// TIA Portal project "Palletizer" (V15.1)

(* hardware
DEVICE "S71500/ET200MP-Station_1"  S7-1500 station
   slot 0: "Profilschiene_0"  6ES7 590-1***0-0AA0
   slot 1: "PLC_1"  CPU 1511-1 PN  6ES7 511-1AK00-0AB0  V1.8
   slot 2: "AI 8xU/I/RTD/TC ST_1"  AI 8xU/I/RTD/TC ST  6ES7 531-7KF00-0AB0  V2.0
   slot 3: "AI 8xU/I/RTD/TC ST_2"  AI 8xU/I/RTD/TC ST  6ES7 531-7KF00-0AB0  V2.0
   slot 4: "AI 8xU/I/RTD/TC ST_3"  AI 8xU/I/RTD/TC ST  6ES7 531-7KF00-0AB0  V2.0
   slot 5: "AI 8xU/I/RTD/TC ST_4"  AI 8xU/I/RTD/TC ST  6ES7 531-7KF00-0AB0  V2.0
   slot 6: "DI 16x24VDC BA_1"  DI 16x24VDC BA  6ES7 521-1BH10-0AA0  V1.0
*)

// ===== PLC "PLC_1"  CPU 1511-1 PN =====

VAR_GLOBAL   // PLC tag table "Standard-Variablentabelle"
   "Pallet at entry" AT %E0.0 : Bool;
   "Clock_Byte" AT %MB0 : Byte;
   "Clock_10Hz" AT %M0.0 : Bool;
   "Clock_5Hz" AT %M0.1 : Bool;
   "Clock_2.5Hz" AT %M0.2 : Bool;
   "Clock_2Hz" AT %M0.3 : Bool;
   "Clock_1.25Hz" AT %M0.4 : Bool;
   "Clock_1Hz" AT %M0.5 : Bool;
   "Clock_0.625Hz" AT %M0.6 : Bool;
   "Clock_0.5Hz" AT %M0.7 : Bool;
   "Pallet at exit" AT %I0.1 : Bool;
   "Pallet loaded" AT %I0.2 : Bool;
   "Box at entry" AT %I0.3 : Bool;
   "Pusher at limit" AT %I0.4 : Bool;
   "Plate limit" AT %I0.5 : Bool;
   "Clamped" AT %I0.6 : Bool;
   "Elevator moving" AT %I0.7 : Bool;
   "Start" AT %I1.0 : Bool;
   "Reset" AT %I1.1 : Bool;
   "Stop" AT %I1.2 : Bool;
   "Emergency stop" AT %I1.3 : Bool;
   "Auto" AT %I1.4 : Bool;
   "Pallet feeder" AT %Q0.0 : Bool;
   "Laod pallet" AT %Q0.1 : Bool;
   "Exit conveyor" AT %Q0.2 : Bool;
   "Move to limit" AT %Q0.3 : Bool;
   "Elevator up" AT %Q0.4 : Bool;
   "Elevator down" AT %Q0.5 : Bool;
   "Box feeder" AT %Q0.6 : Bool;
   "Turn" AT %Q0.7 : Bool;
   "Push" AT %Q1.0 : Bool;
   "Load belt" AT %Q1.1 : Bool;
   "Clamp" AT %Q1.2 : Bool;
   "Open plate" AT %Q1.3 : Bool;
   "Warning light" AT %Q1.4 : Bool;
   "Start light" AT %Q1.5 : Bool;
   "Reset light" AT %Q1.6 : Bool;
   "Stop light" AT %Q1.7 : Bool;
   "Counter" AT %QD30 : DInt;
END_VAR

TYPE "statusCiclo"
   STRUCT
      EmAutomatico : Bool;
      EmManual : Bool;
      CicloIniciado : Bool;
      EmAnomalia : Bool;
      EmEmergencia : Bool;
      EmParada : Bool;
      Reset : Bool;
      AddCont : DInt;
   END_STRUCT;
END_TYPE

TYPE "Controle_Caixas"
   STRUCT
      N_Caixas : Int;
      N_Atingido : Bool;
      Solicitacao_Box : Bool;
      Reset_N_Caixas : Bool;
      Aux_Ordenacao : Bool;
      Ordenado : Bool;
   END_STRUCT;
END_TYPE

// folder: Paletizador

DATA_BLOCK "Painel_DB"   // DB1
{ S7_Optimized_Access := 'TRUE' }
VERSION : 0.1
// stored: InstanceOfName Painel
"Painel"
BEGIN
END_DATA_BLOCK

DATA_BLOCK "Pallet_Feeder_DB"   // DB2
{ S7_Optimized_Access := 'TRUE' }
VERSION : 0.1
// stored: InstanceOfName Pallet_Feeder
"Pallet_Feeder"
BEGIN
END_DATA_BLOCK

DATA_BLOCK "Status"   // DB3
{ S7_Optimized_Access := 'TRUE' }
VERSION : 0.1
BEGIN
END_DATA_BLOCK

DATA_BLOCK "Remove_Pallet_DB"   // DB4
{ S7_Optimized_Access := 'TRUE' }
VERSION : 0.1
// stored: InstanceOfName Remove_Pallet
"Remove_Pallet"
BEGIN
END_DATA_BLOCK

DATA_BLOCK "Box_Feeder_DB"   // DB5
{ S7_Optimized_Access := 'TRUE' }
VERSION : 0.1
// stored: InstanceOfName Box_Feeder
"Box_Feeder"
BEGIN
END_DATA_BLOCK

DATA_BLOCK "Elevador_DB"   // DB6
{ S7_Optimized_Access := 'TRUE' }
VERSION : 0.1
// stored: InstanceOfName Elevador
"Elevador"
BEGIN
END_DATA_BLOCK

DATA_BLOCK "Organizador_DB"   // DB7
{ S7_Optimized_Access := 'TRUE' }
VERSION : 0.1
// stored: InstanceOfName Organizador
"Organizador"
BEGIN
END_DATA_BLOCK

// folder: Paletizador/Organizador

DATA_BLOCK "Orientacao_2_DB"   // DB8
{ S7_Optimized_Access := 'TRUE' }
VERSION : 0.1
// stored: InstanceOfName Orientacao_2
"Orientacao_2"
BEGIN
END_DATA_BLOCK

DATA_BLOCK "Orientacao_1_DB"   // DB10
{ S7_Optimized_Access := 'TRUE' }
VERSION : 0.1
// stored: InstanceOfName Orientacao_1
"Orientacao_1"
BEGIN
END_DATA_BLOCK

// folder: System blocks/Program resources

DATA_BLOCK "Contadir_Camadas"   // DB9
{ S7_Optimized_Access := 'TRUE' }
AUTHOR : Simatic
FAMILY : IEC
NAME : CNTR
VERSION : 1.0
// stored: InstanceOfName IEC_COUNTER
"IEC_COUNTER"
BEGIN
END_DATA_BLOCK

DATA_BLOCK "Contador_Caixas"   // DB11
{ S7_Optimized_Access := 'TRUE' }
AUTHOR : Simatic
FAMILY : IEC
NAME : CNTR
VERSION : 1.0
// stored: InstanceOfName IEC_COUNTER
"IEC_COUNTER"
BEGIN
END_DATA_BLOCK

DATA_BLOCK "Timer_Load_Belt"   // DB13
{ S7_Optimized_Access := 'TRUE' }
AUTHOR : Simatic
FAMILY : IEC
NAME : IEC_TMR
VERSION : 1.0
// stored: InstanceOfName IEC_TIMER
"IEC_TIMER"
BEGIN
END_DATA_BLOCK

DATA_BLOCK "Counter_Push"   // DB14
{ S7_Optimized_Access := 'TRUE' }
AUTHOR : Simatic
FAMILY : IEC
NAME : CNTR
VERSION : 1.0
// stored: InstanceOfName IEC_COUNTER
"IEC_COUNTER"
BEGIN
END_DATA_BLOCK

DATA_BLOCK "Ton_Reset_Push"   // DB15
{ S7_Optimized_Access := 'TRUE' }
AUTHOR : Simatic
FAMILY : IEC
NAME : IEC_TMR
VERSION : 1.0
// stored: InstanceOfName IEC_TIMER
"IEC_TIMER"
BEGIN
END_DATA_BLOCK

DATA_BLOCK "Timer_Clamp"   // DB16
{ S7_Optimized_Access := 'TRUE' }
AUTHOR : Simatic
FAMILY : IEC
NAME : IEC_TMR
VERSION : 1.0
// stored: InstanceOfName IEC_TIMER
"IEC_TIMER"
BEGIN
END_DATA_BLOCK

DATA_BLOCK "Timer_Desce"   // DB17
{ S7_Optimized_Access := 'TRUE' }
AUTHOR : Simatic
FAMILY : IEC
NAME : IEC_TMR
VERSION : 1.0
// stored: InstanceOfName IEC_TIMER
"IEC_TIMER"
BEGIN
END_DATA_BLOCK

// folder: (top level)

FUNCTION "MHJ-PLC-Lab-Function-S71500" : Void   // FC9000, SCL
{ S7_Optimized_Access := 'TRUE' }
VERSION : 0.1
   VAR_TEMP
      Value : Byte;
      ForCounter : Int;
   END_VAR
   VAR CONSTANT
      Value_01_DW : DWord := 16#1223_5486;
      Value_02_DW : DWord := 16#A6C9_D1F5;
   END_VAR
BEGIN

   #Value:=PEEK(area := 16#82,
        dbNumber := 0,
        byteOffset := 511);
   #Value := #Value + 1;

   POKE(area := 16#82,
        dbNumber := 0,
        byteOffset := 511,
        value := #Value);

   POKE(area := 16#82,
        dbNumber := 0,
        byteOffset := 1016,
        value := #Value_01_DW);
   POKE(area := 16#82,
        dbNumber := 0,
        byteOffset := 1020,
        value := #Value_02_DW);

   FOR #ForCounter := 0 TO 63 DO
       #Value:=PEEK(area := 16#1,
            dbNumber := 0,
            byteOffset := #ForCounter);
       POKE(area := 16#81,
            dbNumber := 0,
            byteOffset := #ForCounter,
            value := #Value);
   END_FOR;
   #Value := PEEK(area := 16#1,
                  dbNumber := 0,
                  byteOffset := 512);
   POKE(area := 16#82,
        dbNumber := 0,
        byteOffset := 512,
        value := #Value);
END_FUNCTION

ORGANIZATION_BLOCK "Main"   // OB1, FBD, ProgramCycle
TITLE = "Main Program Sweep (Cycle)"
{ S7_Optimized_Access := 'TRUE' }
VERSION : 0.1
   VAR_INPUT
      Initial_Call : Bool;   // Initial call of this OB
      Remanence : Bool;   // =True, if remanent data are available
   END_VAR
BEGIN

REGION Network 1
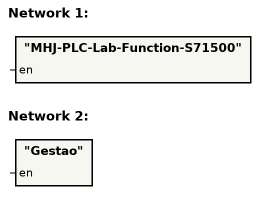
   "MHJ-PLC-Lab-Function-S71500"();
END_REGION

REGION Network 2
   "Gestao"();
END_REGION
END_ORGANIZATION_BLOCK

// folder: Paletizador

FUNCTION "Gestao" : Void   // FC1, LAD
{ S7_Optimized_Access := 'TRUE' }
VERSION : 0.1
BEGIN

REGION Network 1
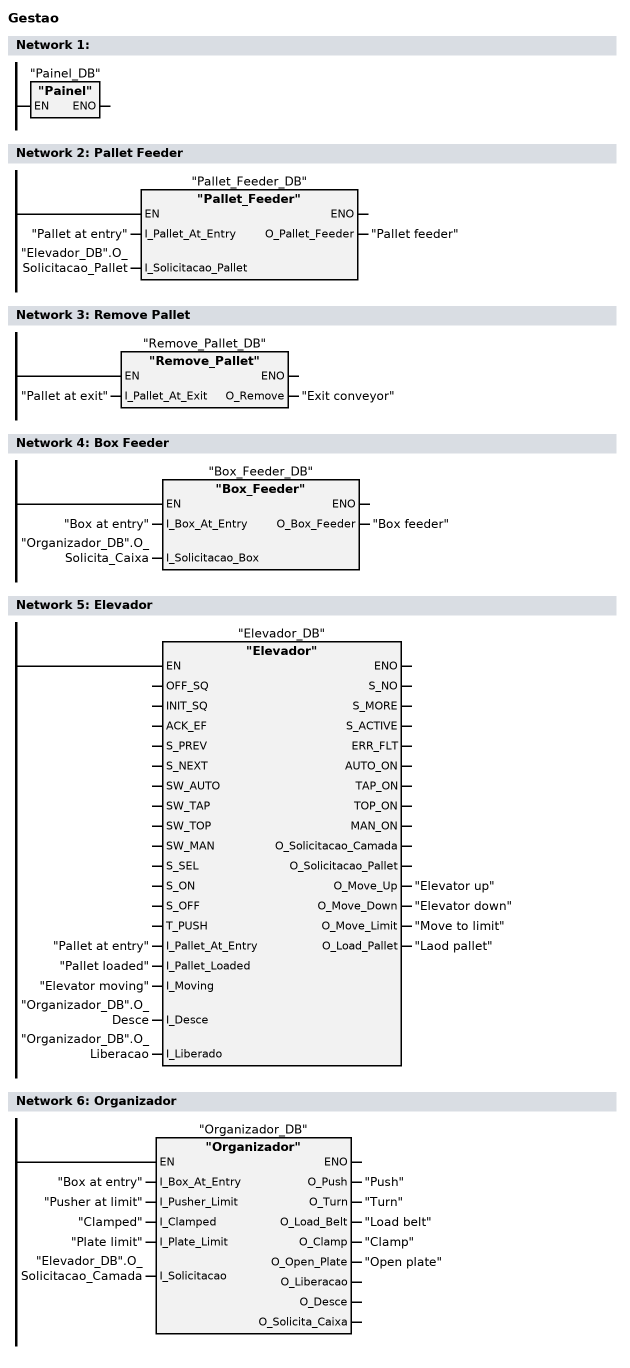
   RUNG wire#powerrail
      "Painel_DB"()
   END_RUNG
   // the same network as SCL:
   "Painel_DB"();   // "Painel"
END_REGION

REGION Network 2: Pallet Feeder
   RUNG wire#powerrail
      "Pallet_Feeder_DB"(I_Pallet_At_Entry := "Pallet at entry", I_Solicitacao_Pallet := "Elevador_DB".O_Solicitacao_Pallet, O_Pallet_Feeder => "Pallet feeder")
   END_RUNG
   // the same network as SCL:
   "Pallet_Feeder_DB"(I_Pallet_At_Entry := "Pallet at entry",   // "Pallet_Feeder"
                      I_Solicitacao_Pallet := "Elevador_DB".O_Solicitacao_Pallet,
                      O_Pallet_Feeder => "Pallet feeder");
END_REGION

REGION Network 3: Remove Pallet
   RUNG wire#powerrail
      "Remove_Pallet_DB"(I_Pallet_At_Exit := "Pallet at exit", O_Remove => "Exit conveyor")
   END_RUNG
   // the same network as SCL:
   "Remove_Pallet_DB"(I_Pallet_At_Exit := "Pallet at exit", O_Remove => "Exit conveyor");   // "Remove_Pallet"
END_REGION

REGION Network 4: Box Feeder
   RUNG wire#powerrail
      "Box_Feeder_DB"(I_Box_At_Entry := "Box at entry", I_Solicitacao_Box := "Organizador_DB".O_Solicita_Caixa, O_Box_Feeder => "Box feeder")
   END_RUNG
   // the same network as SCL:
   "Box_Feeder_DB"(I_Box_At_Entry := "Box at entry",   // "Box_Feeder"
                   I_Solicitacao_Box := "Organizador_DB".O_Solicita_Caixa,
                   O_Box_Feeder => "Box feeder");
END_REGION

REGION Network 5: Elevador
   RUNG wire#powerrail
      "Elevador_DB"(OFF_SQ :=, INIT_SQ :=, ACK_EF :=, S_PREV :=, S_NEXT :=, SW_AUTO :=, SW_TAP :=, SW_TOP :=, SW_MAN :=, S_SEL :=, S_ON :=, S_OFF :=, T_PUSH :=, I_Pallet_At_Entry := "Pallet at entry", I_Pallet_Loaded := "Pallet loaded", I_Moving := "Elevator moving", I_Desce := "Organizador_DB".O_Desce, I_Liberado := "Organizador_DB".O_Liberacao, S_NO =>, S_MORE =>, S_ACTIVE =>, ERR_FLT =>, AUTO_ON =>, TAP_ON =>, TOP_ON =>, MAN_ON =>, O_Solicitacao_Camada =>, O_Solicitacao_Pallet =>, O_Move_Up => "Elevator up", O_Move_Down => "Elevator down", O_Move_Limit => "Move to limit", O_Load_Pallet => "Laod pallet")
   END_RUNG
   // the same network as SCL:
   "Elevador_DB"(I_Pallet_At_Entry := "Pallet at entry",   // "Elevador"
                 I_Pallet_Loaded := "Pallet loaded",
                 I_Moving := "Elevator moving",
                 I_Desce := "Organizador_DB".O_Desce,
                 I_Liberado := "Organizador_DB".O_Liberacao,
                 O_Move_Up => "Elevator up",
                 O_Move_Down => "Elevator down",
                 O_Move_Limit => "Move to limit",
                 O_Load_Pallet => "Laod pallet");
END_REGION

REGION Network 6: Organizador
   RUNG wire#powerrail
      "Organizador_DB"(I_Box_At_Entry := "Box at entry", I_Pusher_Limit := "Pusher at limit", I_Clamped := "Clamped", I_Plate_Limit := "Plate limit", I_Solicitacao := "Elevador_DB".O_Solicitacao_Camada, O_Push => "Push", O_Turn => "Turn", O_Load_Belt => "Load belt", O_Clamp => "Clamp", O_Open_Plate => "Open plate", O_Liberacao =>, O_Desce =>, O_Solicita_Caixa =>)
   END_RUNG
   // the same network as SCL:
   "Organizador_DB"(I_Box_At_Entry := "Box at entry",   // "Organizador"
                    I_Pusher_Limit := "Pusher at limit",
                    I_Clamped := "Clamped",
                    I_Plate_Limit := "Plate limit",
                    I_Solicitacao := "Elevador_DB".O_Solicitacao_Camada,
                    O_Push => "Push",
                    O_Turn => "Turn",
                    O_Load_Belt => "Load belt",
                    O_Clamp => "Clamp",
                    O_Open_Plate => "Open plate");
END_REGION
END_FUNCTION

// folder: Paletizador/Box_Feeder

FUNCTION_BLOCK "Box_Feeder"   // FB4, LAD
{ S7_Optimized_Access := 'TRUE' }
VERSION : 0.1
   VAR_INPUT
      I_Box_At_Entry : Bool;
      I_Solicitacao_Box : Bool;
   END_VAR
   VAR_OUTPUT
      O_Box_Feeder : Bool;
   END_VAR
BEGIN

REGION Network 1: Em Automatico
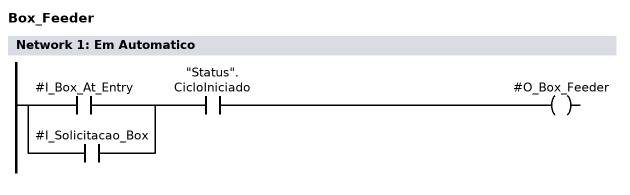
   RUNG wire#powerrail
      Contact( #I_Box_At_Entry )
      wire#w1
      Contact( "Status".CicloIniciado )
      Coil( #O_Box_Feeder )
   END_RUNG
   RUNG wire#powerrail
      Contact( #I_Solicitacao_Box )
   END_RUNG wire#w1
   // the same network as SCL:
   #O_Box_Feeder := (#I_Box_At_Entry OR #I_Solicitacao_Box) AND "Status".CicloIniciado;
END_REGION
END_FUNCTION_BLOCK

// folder: Paletizador/Elevador

FUNCTION_BLOCK "Elevador"   // FB6, GRAPH_PLUS
{ S7_Optimized_Access := 'TRUE' }
VERSION : 0.1
   VAR_INPUT
      OFF_SQ : Bool := false;   // Turn sequence off
      INIT_SQ : Bool := false;   // Set sequence to initial state
      ACK_EF : Bool := false;   // Acknowledge all errors and faults
      S_PREV : Bool := false;   // Output previous step in parameter S_NO
      S_NEXT : Bool := false;   // Indicate next step in parameter S_NO
      SW_AUTO : Bool := false;   // Automatic mode
      SW_TAP : Bool := false;   // Semiautomatic/switch with transition
      SW_TOP : Bool := false;   // Semiautomatic/ignore transition
      SW_MAN : Bool := false;   // Manual mode
      S_SEL : Int := 0;   // Select step to be output to S_NO
      S_ON : Bool := false;   // Activate step indicated in S_NO
      S_OFF : Bool := false;   // Deactivate step indicated S_NO
      T_PUSH : Bool := false;   // Enable transition to switch in semi automatic mode
      I_Pallet_At_Entry : Bool;
      I_Pallet_Loaded : Bool;
      I_Moving : Bool;
      I_Desce : Bool;
      I_Liberado : Bool;
   END_VAR
   VAR_OUTPUT
      S_NO : Int := 0;   // Step number
      S_MORE : Bool := false;   // More steps are available and can be shown in S_NO
      S_ACTIVE : Bool := false;   // Step indicated in S_NO is active
      ERR_FLT : Bool := false;   // Interlock or supervision group error
      AUTO_ON : Bool := false;   // Automatic mode is active
      TAP_ON : Bool := false;   // Semiautomatic mode/step with transition enabled
      TOP_ON : Bool := false;   // Semiautomatic mode/ignore transition enabled
      MAN_ON : Bool := false;   // Manual mode is active
      O_Solicitacao_Camada : Bool;
      O_Solicitacao_Pallet : Bool;
      O_Move_Up : Bool;
      O_Move_Down : Bool;
      O_Move_Limit : Bool;
      O_Load_Pallet : Bool;
   END_VAR
   VAR
      HMI_INFO : Array[0..8] of UInt;
      IF_PAR : G7_IfParPlus_V2;
      RT_DATA : G7_RTDataPlus_V2;   // Internal data area
      Trans5 : G7_TransitionPlus_V2;   // Transition structure
      Trans1 : G7_TransitionPlus_V2;   // Transition structure
      Trans2 : G7_TransitionPlus_V2;   // Transition structure
      Trans3 : G7_TransitionPlus_V2;   // Transition structure
      Trans6 : G7_TransitionPlus_V2;   // Transition structure
      Trans7 : G7_TransitionPlus_V2;   // Transition structure
      Trans8 : G7_TransitionPlus_V2;   // Transition structure
      Trans9 : G7_TransitionPlus_V2;   // Transition structure
      Trans10 : G7_TransitionPlus_V2;   // Transition structure
      Wainting : G7_StepPlus_V2;   // Step structure
      Home : G7_StepPlus_V2;   // Step structure
      "Carrega pallet" : G7_StepPlus_V2;   // Step structure
      Sobe : G7_StepPlus_V2;   // Step structure
      "Solicita Caixas" : G7_StepPlus_V2;   // Step structure
      Step6 : G7_StepPlus_V2;   // Step structure
      Step7 : G7_StepPlus_V2;   // Step structure
      Step8 : G7_StepPlus_V2;   // Step structure
      SINI : Array[0..1] of USInt;
      LSTT : Array[0..8] of USInt;
      ATAJ : Array[0..8] of USInt;
      ATAB : Array[0..8] of USInt;
      PSTT : Array[0..8] of USInt;
      NSTT : Array[0..8] of USInt;
      ASSJ : Array[0..7] of USInt;
      ASSB : Array[0..7] of USInt;
      PTTS : Array[0..7] of USInt;
      NTTS : Array[0..7] of USInt;
      SW_SQTS : Array[0..7] of USInt;
      SWITCH : Array[0..1] of USInt;
      TVX : Array[0..3] of USInt;
      TTX : Array[0..3] of USInt;
      TSX : Array[0..1] of USInt;
      S00X : Array[0..1] of USInt;
      SOFFX : Array[0..1] of USInt;
      SONX : Array[0..1] of USInt;
      SAX : Array[0..1] of USInt;
      SERRX : Array[0..8] of USInt;
      SMX : Array[0..8] of USInt;
      S0X : Array[0..8] of USInt;
      S1X : Array[0..8] of USInt;
      IL_ALARM_INST : Program_Alarm;
      SUP_ALARM_INST : Program_Alarm;
      STEP_TIME_ALARM_INST : Program_Alarm;
      IEC_TIMER_INST : IEC_TIMER;
      TRANSACTION_FLAG : Bool := false;
   END_VAR
   // SINI[0] := 2;
   // LSTT[0] := 255;
   // LSTT[1] := 255;
   // ATAJ[1] := 1;
   // ATAJ[2] := 2;
   // ATAB[1] := 1;
   // ATAB[2] := 2;
   // PSTT[1] := 1;
   // PSTT[2] := 2;
   // NSTT[0] := 1;
   // NSTT[1] := 2;
   // ASSJ[1] := 1;
   // ASSJ[2] := 2;
   // ASSB[1] := 1;
   // ASSB[2] := 2;
   // PTTS[0] := 255;
   // PTTS[2] := 1;
   // NTTS[1] := 1;
   // NTTS[2] := 2;
   // TVX[0] := 16#1;
   // TTX[0] := 16#1;
   // TSX[0] := 16#1;
   // S00X[0] := 16#1;
   // SOFFX[0] := 16#1;
   // SONX[0] := 16#1;
   // SAX[0] := 16#1;
   // SERRX[0] := 16#1;
   // SMX[0] := 16#1;
   // S0X[0] := 16#1;
   // S1X[0] := 16#1;
   // LSTT[2] := 255;
   // ATAJ[3] := 3;
   // ATAB[3] := 3;
   // PSTT[3] := 3;
   // NSTT[2] := 3;
   // ASSJ[3] := 3;
   // ASSB[3] := 3;
   // PTTS[3] := 2;
   // NTTS[3] := 3;
   // LSTT[4] := 255;
   // ATAJ[4] := 4;
   // ATAB[4] := 5;
   // PSTT[4] := 4;
   // NSTT[4] := 6;
   // ASSJ[4] := 4;
   // ASSB[4] := 4;
   // PTTS[4] := 3;
   // NTTS[4] := 5;
   // LSTT[3] := 255;
   // LSTT[5] := 255;
   // LSTT[6] := 255;
   // ATAJ[5] := 5;
   // ATAJ[6] := 6;
   // ATAB[5] := 4;
   // ATAB[6] := 6;
   // PSTT[5] := 4;
   // PSTT[6] := 5;
   // NSTT[3] := 4;
   // NSTT[5] := 5;
   // NSTT[6] := 255;
   // ASSJ[5] := 5;
   // ASSB[5] := 5;
   // PTTS[5] := 5;
   // NTTS[5] := 6;
   // SW_SQTS[5] := 1;
   // LSTT[7] := 255;
   // ATAJ[7] := 7;
   // ATAB[7] := 7;
   // PSTT[7] := 6;
   // NSTT[7] := 7;
   // ASSJ[6] := 6;
   // ASSB[6] := 6;
   // PTTS[6] := 4;
   // NTTS[6] := 7;
   // SW_SQTS[6] := 2;
   // LSTT[8] := 255;
   // ATAJ[8] := 8;
   // ATAB[8] := 8;
   // PSTT[8] := 7;
   // NSTT[8] := 255;
   // ASSJ[7] := 7;
   // ASSB[7] := 7;
   // PTTS[7] := 7;
   // NTTS[7] := 8;
   // SW_SQTS[7] := 2;
BEGIN
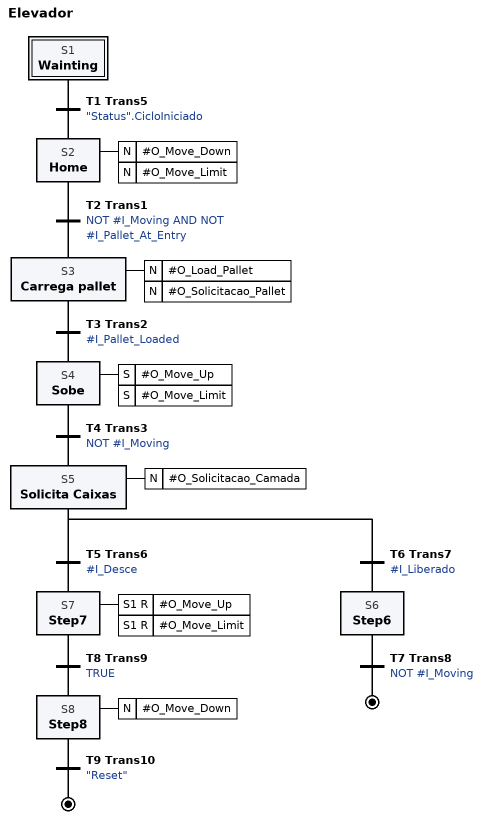
   // sequencer 1
   INITIAL_STEP Wainting:   // S1, max time T#10S, warning time T#7S
   END_STEP
   TRANSITION Trans5 FROM Wainting TO Home   // T1
      := "Status".CicloIniciado;
   END_TRANSITION
   STEP "Carrega pallet":   // S3, max time T#10S, warning time T#7S
              N    #O_Load_Pallet
              N    #O_Solicitacao_Pallet
   END_STEP
   TRANSITION Trans2 FROM "Carrega pallet" TO Sobe   // T3
      := #I_Pallet_Loaded;
   END_TRANSITION
   STEP Sobe:   // S4, max time T#10S, warning time T#7S
              S    #O_Move_Up
              S    #O_Move_Limit
   END_STEP
   TRANSITION Trans3 FROM Sobe TO "Solicita Caixas"   // T4
      := NOT #I_Moving;
   END_TRANSITION
   STEP "Solicita Caixas":   // S5, max time T#10S, warning time T#7S
              N    #O_Solicitacao_Camada
   END_STEP
   TRANSITION Trans6 FROM "Solicita Caixas" TO Step7   // T5
      := #I_Desce;
   END_TRANSITION
   TRANSITION Trans7 FROM "Solicita Caixas" TO Step6   // T6
      := #I_Liberado;
   END_TRANSITION
   STEP Home:   // S2, max time T#10S, warning time T#7S
              N    #O_Move_Down
              N    #O_Move_Limit
   END_STEP
   TRANSITION Trans1 FROM Home TO "Carrega pallet"   // T2
      := NOT #I_Moving AND NOT #I_Pallet_At_Entry;
   END_TRANSITION
   STEP Step6:   // S6, max time T#10S, warning time T#7S
   END_STEP
   TRANSITION Trans8 FROM Step6 TO END   // T7
      := NOT #I_Moving;
   END_TRANSITION
   STEP Step7:   // S7, max time T#10S, warning time T#7S
          S1  R    #O_Move_Up
          S1  R    #O_Move_Limit
   END_STEP
   TRANSITION Trans9 FROM Step7 TO Step8   // T8
      := TRUE;
   END_TRANSITION
   STEP Step8:   // S8, max time T#10S, warning time T#7S
              N    #O_Move_Down
   END_STEP
   TRANSITION Trans10 FROM Step8 TO END   // T9
      := "Reset";
   END_TRANSITION
END_FUNCTION_BLOCK

// folder: Paletizador/Organizador

FUNCTION_BLOCK "Organizador"   // FB5, LAD
{ S7_Optimized_Access := 'TRUE' }
VERSION : 0.1
   VAR_INPUT
      I_Box_At_Entry : Bool;
      I_Pusher_Limit : Bool;
      I_Clamped : Bool;
      I_Plate_Limit : Bool;
      I_Solicitacao : Bool;
   END_VAR
   VAR_OUTPUT
      O_Push : Bool;
      O_Turn : Bool;
      O_Load_Belt : Bool;
      O_Clamp : Bool;
      O_Open_Plate : Bool;
      O_Liberacao : Bool;
      O_Desce : Bool;
      O_Solicita_Caixa : Bool;
   END_VAR
   VAR
      M1 : Bool;
      M2 : Bool;
      M3 : Bool;
      SetTurn : Bool;
      Local_Reset : Bool;
      Push_1 : Bool;
      Push_2 : Bool;
      Caixa_1 : Bool;
      Caixa_2 : Bool;
      Soli_caixa : Bool;
      Alvo_Camadas : Int := 4;
      CV_Camadas : Int;
      Controle_Camadas : Int;
      Layer_Shift : Bool;
      delay_Plate : Bool;
   END_VAR
   VAR_TEMP   // added for the SCL form of the ladder/FBD networks
      _w1 : Bool;
   END_VAR
BEGIN

REGION Network 1: Solicitação Caixa
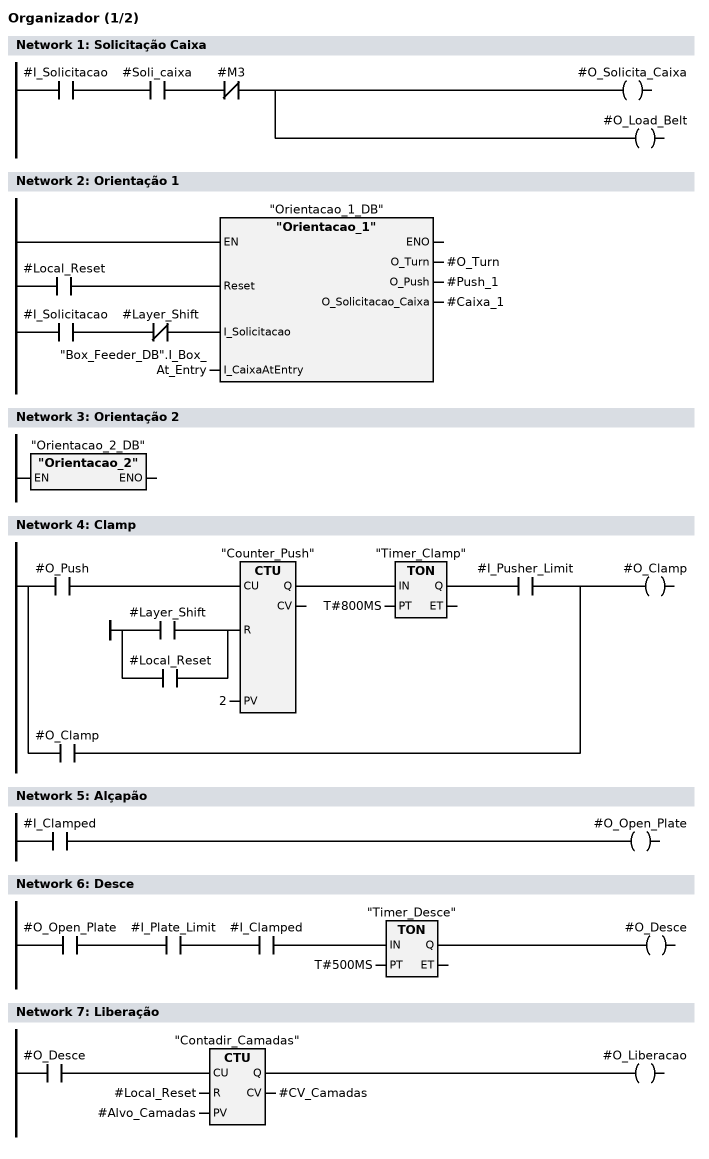
   RUNG wire#powerrail
      Contact( #I_Solicitacao )
      Contact( #Soli_caixa )
      I_Contact( #M3 )
      wire#w1
      Coil( #O_Solicita_Caixa )
   END_RUNG
   RUNG wire#w1
      Coil( #O_Load_Belt )
   END_RUNG
   // the same network as SCL:
   #O_Solicita_Caixa := #I_Solicitacao AND #Soli_caixa AND NOT #M3;
   #O_Load_Belt := #O_Solicita_Caixa;
END_REGION

REGION Network 2: Orientação 1
   RUNG wire#powerrail
      "Orientacao_1_DB"(Reset := wire#w1, I_Solicitacao := wire#w2, I_CaixaAtEntry := "Box_Feeder_DB".I_Box_At_Entry, O_Turn => #O_Turn, O_Push => #Push_1, O_Solicitacao_Caixa => #Caixa_1)
   END_RUNG
   RUNG wire#powerrail
      Contact( #Local_Reset )
   END_RUNG wire#w1
   RUNG wire#powerrail
      Contact( #I_Solicitacao )
      I_Contact( #Layer_Shift )
   END_RUNG wire#w2
   // the same network as SCL:
   "Orientacao_1_DB"(Reset := #Local_Reset,   // "Orientacao_1"
                     I_Solicitacao := #I_Solicitacao AND NOT #Layer_Shift,
                     I_CaixaAtEntry := "Box_Feeder_DB".I_Box_At_Entry,
                     O_Turn => #O_Turn,
                     O_Push => #Push_1,
                     O_Solicitacao_Caixa => #Caixa_1);
END_REGION

REGION Network 3: Orientação 2
   RUNG wire#powerrail
      "Orientacao_2_DB"()
   END_RUNG
   // the same network as SCL:
   "Orientacao_2_DB"();   // "Orientacao_2"
END_REGION

REGION Network 4: Clamp
   "Counter_Push".CTU(CU := #O_Push, R := #Layer_Shift OR #Local_Reset, PV := 2);
   "Timer_Clamp".TON(IN := "Counter_Push".Q, PT := T#800MS);
   #O_Clamp := ("Timer_Clamp".Q AND #I_Pusher_Limit) OR #O_Clamp;
END_REGION

REGION Network 5: Alçapão
   RUNG wire#powerrail
      Contact( #I_Clamped )
      Coil( #O_Open_Plate )
   END_RUNG
   // the same network as SCL:
   #O_Open_Plate := #I_Clamped;
END_REGION

REGION Network 6: Desce
   "Timer_Desce".TON(IN := #O_Open_Plate AND #I_Plate_Limit AND #I_Clamped, PT := T#500MS);
   #O_Desce := "Timer_Desce".Q;
END_REGION

REGION Network 7: Liberação
   "Contadir_Camadas".CTU(CU := #O_Desce, R := #Local_Reset, PV := #Alvo_Camadas, CV => #CV_Camadas);
   #O_Liberacao := "Contadir_Camadas".Q;
END_REGION

REGION Network 8: Controle de Orientação
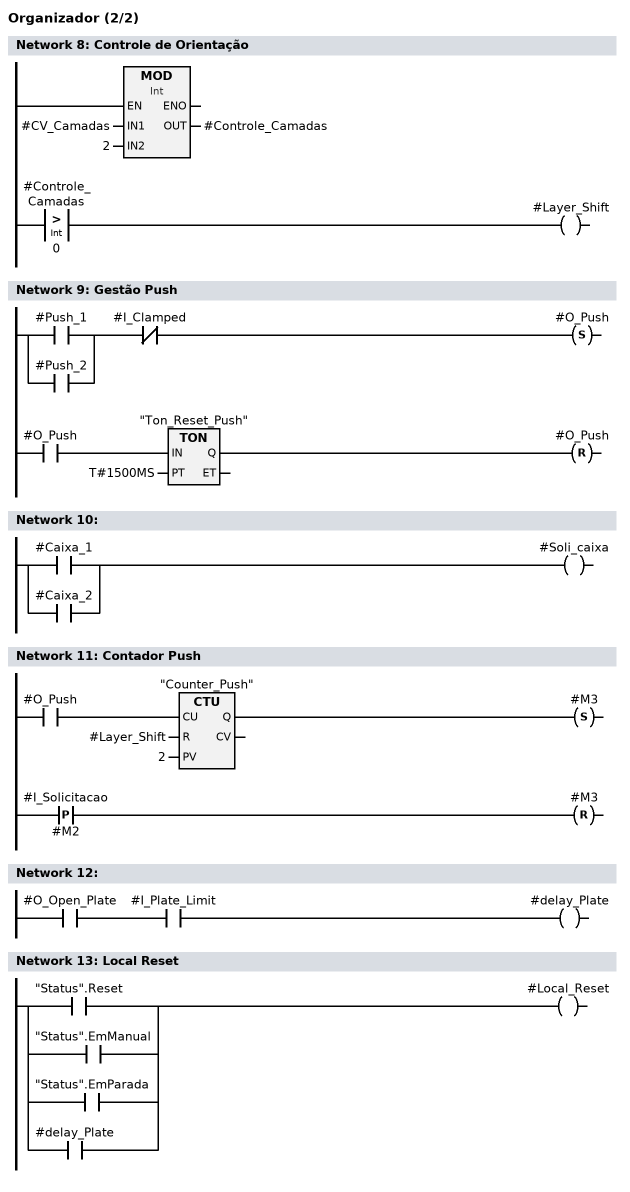
   RUNG wire#powerrail
      { S7_Templates := "SrcType := Int" } Mod(in1 := #CV_Camadas, in2 := 2, out => #Controle_Camadas)
   END_RUNG
   RUNG wire#powerrail
      { S7_Templates := "SrcType := Int" } GT_Contact(in1 := #Controle_Camadas, in2 := 0)
      Coil( #Layer_Shift )
   END_RUNG
   // the same network as SCL:
   #Controle_Camadas := #CV_Camadas MOD 2;
   #Layer_Shift := #Controle_Camadas > 0;
END_REGION

REGION Network 9: Gestão Push
   IF (#Push_1 OR #Push_2) AND NOT #I_Clamped THEN #O_Push := TRUE; END_IF;
   "Ton_Reset_Push".TON(IN := #O_Push, PT := T#1500MS);
   IF "Ton_Reset_Push".Q THEN #O_Push := FALSE; END_IF;
END_REGION

REGION Network 10
   RUNG wire#powerrail
      Contact( #Caixa_1 )
      wire#w1
      Coil( #Soli_caixa )
   END_RUNG
   RUNG wire#powerrail
      Contact( #Caixa_2 )
   END_RUNG wire#w1
   // the same network as SCL:
   #Soli_caixa := #Caixa_1 OR #Caixa_2;
END_REGION

REGION Network 11: Contador Push
   "Counter_Push".CTU(CU := #O_Push, R := #Layer_Shift, PV := 2);
   IF "Counter_Push".Q THEN #M3 := TRUE; END_IF;
   #_w1 := #I_Solicitacao AND NOT #M2;   // rising edge of #I_Solicitacao
   #M2 := #I_Solicitacao;
   IF #_w1 THEN #M3 := FALSE; END_IF;
END_REGION

REGION Network 12
   RUNG wire#powerrail
      Contact( #O_Open_Plate )
      Contact( #I_Plate_Limit )
      Coil( #delay_Plate )
   END_RUNG
   // the same network as SCL:
   #delay_Plate := #O_Open_Plate AND #I_Plate_Limit;
END_REGION

REGION Network 13: Local Reset
   RUNG wire#powerrail
      Contact( "Status".Reset )
      wire#w1
      Coil( #Local_Reset )
   END_RUNG
   RUNG wire#powerrail
      Contact( "Status".EmManual )
   END_RUNG wire#w1
   RUNG wire#powerrail
      Contact( "Status".EmParada )
   END_RUNG wire#w1
   RUNG wire#powerrail
      Contact( #delay_Plate )
   END_RUNG wire#w1
   // the same network as SCL:
   #Local_Reset := "Status".Reset OR "Status".EmManual OR "Status".EmParada OR #delay_Plate;
END_REGION
END_FUNCTION_BLOCK

// folder: Paletizador/Organizador/Orientacoes

FUNCTION_BLOCK "Orientacao_1"   // FB7, LAD
{ S7_Optimized_Access := 'TRUE' }
VERSION : 0.1
   VAR_INPUT
      Reset : Bool;
      I_Solicitacao : Bool;
      I_CaixaAtEntry : Bool;
   END_VAR
   VAR_OUTPUT
      O_Turn : Bool;
      O_Push : Bool;
      O_Solicitacao_Caixa : Bool;
   END_VAR
   VAR
      M1 : Bool;
      M2 : Bool;
      N_Atingido : Bool;
      Push : Bool;
      Load_Lock : Bool;
   END_VAR
   VAR_TEMP   // added for the SCL form of the ladder/FBD networks
      _w1 : Bool;
      _w2 : Bool;
   END_VAR
BEGIN

REGION Network 1: Gestão Turn
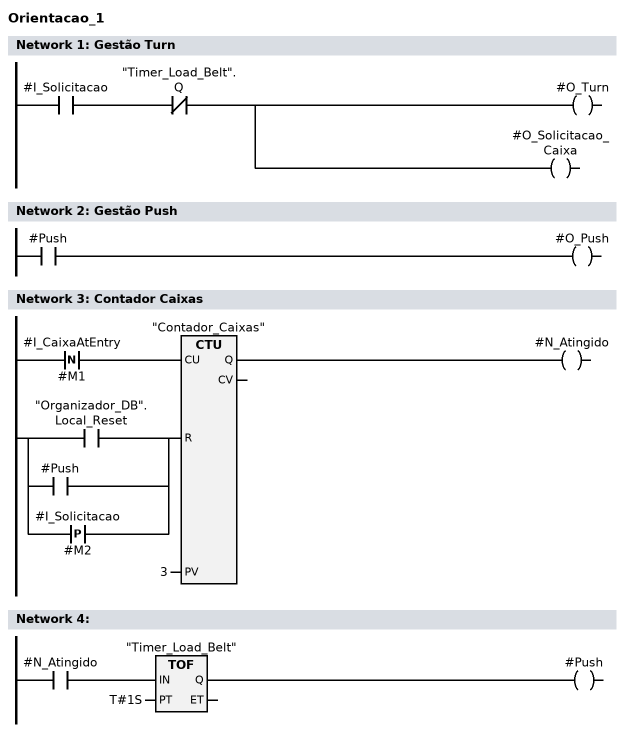
   RUNG wire#powerrail
      Contact( #I_Solicitacao )
      I_Contact( "Timer_Load_Belt".Q )
      wire#w1
      Coil( #O_Turn )
   END_RUNG
   RUNG wire#w1
      Coil( #O_Solicitacao_Caixa )
   END_RUNG
   // the same network as SCL:
   #O_Turn := #I_Solicitacao AND NOT "Timer_Load_Belt".Q;
   #O_Solicitacao_Caixa := #O_Turn;
END_REGION

REGION Network 2: Gestão Push
   RUNG wire#powerrail
      Contact( #Push )
      Coil( #O_Push )
   END_RUNG
   // the same network as SCL:
   #O_Push := #Push;
END_REGION

REGION Network 3: Contador Caixas
   #_w1 := NOT #I_CaixaAtEntry AND #M1;   // falling edge of #I_CaixaAtEntry
   #M1 := #I_CaixaAtEntry;
   #_w2 := #I_Solicitacao AND NOT #M2;   // rising edge of #I_Solicitacao
   #M2 := #I_Solicitacao;
   "Contador_Caixas".CTU(CU := #_w1, R := "Organizador_DB".Local_Reset OR #Push OR #_w2, PV := 3);
   #N_Atingido := "Contador_Caixas".Q;
END_REGION

REGION Network 4
   "Timer_Load_Belt".TOF(IN := #N_Atingido, PT := T#1S);
   #Push := "Timer_Load_Belt".Q;
END_REGION
END_FUNCTION_BLOCK

FUNCTION_BLOCK "Orientacao_2"   // FB8, LAD
{ S7_Optimized_Access := 'TRUE' }
VERSION : 0.1
BEGIN
END_FUNCTION_BLOCK

// folder: Paletizador/Painel_Controle

FUNCTION_BLOCK "Painel"   // FB1, LAD
{ S7_Optimized_Access := 'TRUE' }
VERSION : 0.1
   VAR
      M_Start : Bool;
      M_Stop : Bool;
   END_VAR
   VAR_TEMP   // added for the SCL form of the ladder/FBD networks
      _w1 : Bool;
   END_VAR
BEGIN

REGION Network 1: ############## CONTROLES ##############
END_REGION

REGION Network 2: Start
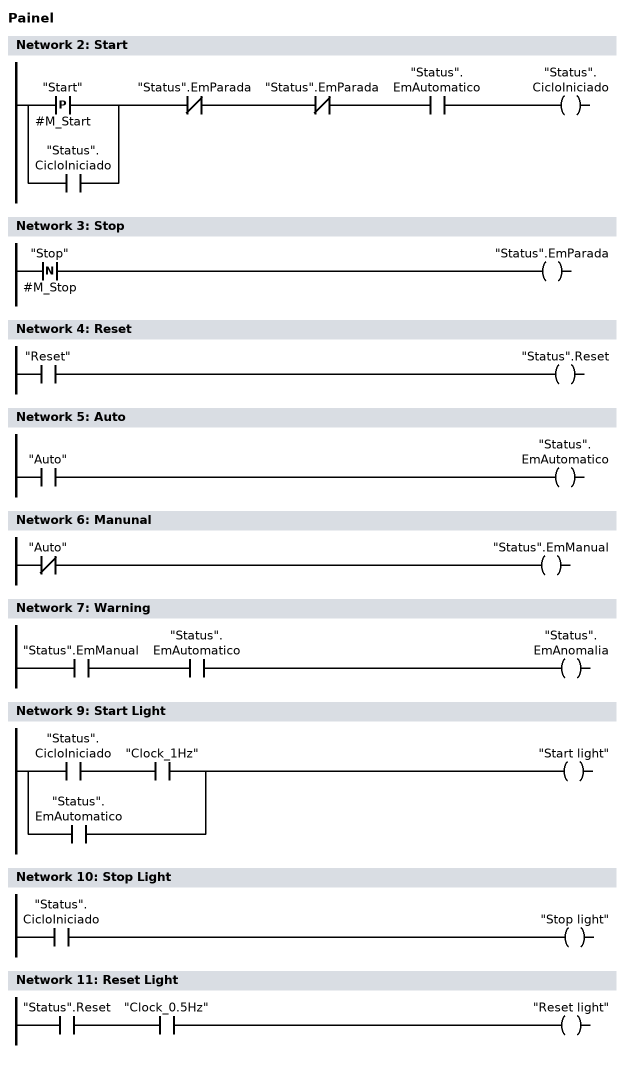
   RUNG wire#powerrail
      P_Contact(operand := "Start", bit := #M_Start)
      wire#w1
      I_Contact( "Status".EmParada )
      I_Contact( "Status".EmParada )
      Contact( "Status".EmAutomatico )
      Coil( "Status".CicloIniciado )
   END_RUNG
   RUNG wire#powerrail
      Contact( "Status".CicloIniciado )
   END_RUNG wire#w1
   // the same network as SCL:
   #_w1 := "Start" AND NOT #M_Start;   // rising edge of "Start"
   #M_Start := "Start";
   "Status".CicloIniciado := (#_w1 OR "Status".CicloIniciado) AND NOT "Status".EmParada AND NOT "Status".EmParada AND "Status".EmAutomatico;
END_REGION

REGION Network 3: Stop
   RUNG wire#powerrail
      N_Contact(operand := "Stop", bit := #M_Stop)
      Coil( "Status".EmParada )
   END_RUNG
   // the same network as SCL:
   #_w1 := NOT "Stop" AND #M_Stop;   // falling edge of "Stop"
   #M_Stop := "Stop";
   "Status".EmParada := #_w1;
END_REGION

REGION Network 4: Reset
   RUNG wire#powerrail
      Contact( "Reset" )
      Coil( "Status".Reset )
   END_RUNG
   // the same network as SCL:
   "Status".Reset := "Reset";
END_REGION

REGION Network 5: Auto
   RUNG wire#powerrail
      Contact( "Auto" )
      Coil( "Status".EmAutomatico )
   END_RUNG
   // the same network as SCL:
   "Status".EmAutomatico := "Auto";
END_REGION

REGION Network 6: Manunal
   RUNG wire#powerrail
      I_Contact( "Auto" )
      Coil( "Status".EmManual )
   END_RUNG
   // the same network as SCL:
   "Status".EmManual := NOT "Auto";
END_REGION

REGION Network 7: Warning
   RUNG wire#powerrail
      Contact( "Status".EmManual )
      Contact( "Status".EmAutomatico )
      Coil( "Status".EmAnomalia )
   END_RUNG
   // the same network as SCL:
   "Status".EmAnomalia := "Status".EmManual AND "Status".EmAutomatico;
END_REGION

REGION Network 8: ############## SINALIZAÇAO ##################
END_REGION

REGION Network 9: Start Light
   RUNG wire#powerrail
      Contact( "Status".CicloIniciado )
      Contact( "Clock_1Hz" )
      wire#w1
      Coil( "Start light" )
   END_RUNG
   RUNG wire#powerrail
      Contact( "Status".EmAutomatico )
   END_RUNG wire#w1
   // the same network as SCL:
   "Start light" := ("Status".CicloIniciado AND "Clock_1Hz") OR "Status".EmAutomatico;
END_REGION

REGION Network 10: Stop Light
   RUNG wire#powerrail
      Contact( "Status".CicloIniciado )
      Coil( "Stop light" )
   END_RUNG
   // the same network as SCL:
   "Stop light" := "Status".CicloIniciado;
END_REGION

REGION Network 11: Reset Light
   RUNG wire#powerrail
      Contact( "Status".Reset )
      Contact( "Clock_0.5Hz" )
      Coil( "Reset light" )
   END_RUNG
   // the same network as SCL:
   "Reset light" := "Status".Reset AND "Clock_0.5Hz";
END_REGION
END_FUNCTION_BLOCK

// folder: Paletizador/Pallet_Feeder

FUNCTION_BLOCK "Pallet_Feeder"   // FB2, LAD
{ S7_Optimized_Access := 'TRUE' }
VERSION : 0.1
   VAR_INPUT
      I_Pallet_At_Entry : Bool;
      I_Solicitacao_Pallet : Bool;
   END_VAR
   VAR_OUTPUT
      O_Pallet_Feeder : Bool;
   END_VAR
BEGIN

REGION Network 1: Em Automatico
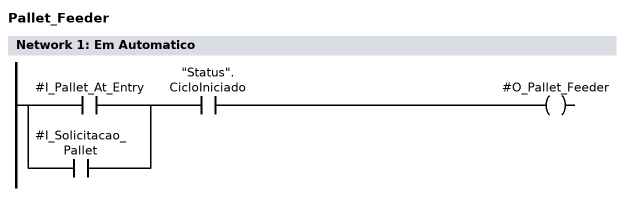
   RUNG wire#powerrail
      Contact( #I_Pallet_At_Entry )
      wire#w1
      Contact( "Status".CicloIniciado )
      Coil( #O_Pallet_Feeder )
   END_RUNG
   RUNG wire#powerrail
      Contact( #I_Solicitacao_Pallet )
   END_RUNG wire#w1
   // the same network as SCL:
   #O_Pallet_Feeder := (#I_Pallet_At_Entry OR #I_Solicitacao_Pallet) AND "Status".CicloIniciado;
END_REGION

REGION Network 2: Em Manual
END_REGION
END_FUNCTION_BLOCK

// folder: Paletizador/Remove_Pallet

FUNCTION_BLOCK "Remove_Pallet"   // FB3, LAD
{ S7_Optimized_Access := 'TRUE' }
VERSION : 0.1
   VAR_INPUT
      I_Pallet_At_Exit : Bool;
   END_VAR
   VAR_OUTPUT
      O_Remove : Bool;
   END_VAR
BEGIN

REGION Network 1: Em Automatico
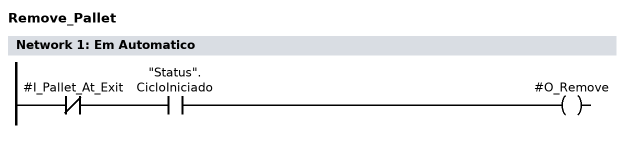
   RUNG wire#powerrail
      I_Contact( #I_Pallet_At_Exit )
      Contact( "Status".CicloIniciado )
      Coil( #O_Remove )
   END_RUNG
   // the same network as SCL:
   #O_Remove := NOT #I_Pallet_At_Exit AND "Status".CicloIniciado;
END_REGION
END_FUNCTION_BLOCK